// SIMATIC S7-200 SMART project (STEP 7-Micro/WIN SMART), CPU ST40

SYMBOL_TABLE Table 1
Motor            Q0.0
ON_SWITCH        I0.0
OFF_SWITCH       I0.1
END_SYMBOL_TABLE

ORGANIZATION_BLOCK MAIN:OB1
TITLE=Program Comments
BEGIN
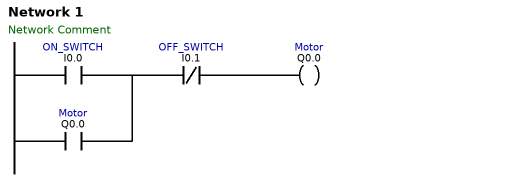
Network 1
// Network Comment
LD     ON_SWITCH:I0.0
O      Motor:Q0.0
AN     OFF_SWITCH:I0.1
=      Motor:Q0.0
END_ORGANIZATION_BLOCK
